{attribute 'qualified_only'}
VAR_GLOBAL

	Test_Axis: Axis; 
	
	RobotVars : Robot;
	
END_VAR

(* stored: Version 1.1.0.1, ProductVersion 3.1.4024.4
   GVL GVL: Id {8e5f239a-c4e9-4a40-a359-44bb19d6c3ee} *)
